// TIA Portal V17 export
// export: Created 2024-08-20T10:59:42.6043051Z, ExportSetting WithDefaults, DisplayName Totally Integrated Automation Portal, DisplayVersion V17 Update 4, DisplayName TIA Portal Openness, DisplayVersion V17 Update 4, DisplayName TIA Portal Version Control Interface, DisplayVersion V17, DisplayName STEP 7 Professional, DisplayVersion V17 Update 4, DisplayName STEP 7 Safety, DisplayVersion V17, DisplayName WinCC Advanced, DisplayVersion V17 Update 4
DATA_BLOCK "Redes"   // DB500
{ S7_Optimized_Access := 'FALSE' }
VERSION : 0.1
// stored: AutoNumber false, DBAccessibleFromOPCUA true, IsOnlyStoredInLoadMemory false, IsWriteProtectedInAS false
   VAR
      "CONNECT-MGE-PCM-E-CF-01" { S7_SetPoint := 'True'} : TCON_IP_v4;   // Dados de configuração
      "CONNECT-MGE-QGBT-AUX-01" { S7_SetPoint := 'True'} : TCON_IP_v4;   // Dados de configuração
      "Register-MGE-PCM-E-CF-01" : Array[0..38] of DInt;   // Tabela para receber os dados
      "Register-MGE-QGBT-AUX-01" : Array[0..38] of DInt;   // Tabela para receber os dados
      LADDR_PROFINET : HW_IOSYSTEM := 261;   // Endereço de hardware
      MODE_PROFINET : UInt := 4;   // Modo de operação da funcção
      RET_VAL_PROFINET : Int;   // Terorno de diagnóstico
      ESTADO_PROFINET : Array[0..1023] of Bool;   // Diagnóstico da rede PROFINET
      DONE_MB : Array[0..60] of Bool;   // Sinaliza fim de execução
      BUSY_MB : Array[0..60] of Bool;   // Sinaliza espera
      ERROR_MB : Array[0..60] of Bool;   // Sinaliza erro
      STATUS_MB : Array[0..60] of Word;   // Satus da comunicação
      START_MB : Array[0..60] of Bool;   // Inicia comunicação
      FCOM_MB : Array[0..60] of Bool;   // Falha de comunicação
      HAB_MB : Array[0..60] of Bool;   // Habilita comunicação MODBUS
      INICIA_MB : Bool;   // INICIA CICLO DE COMUNICAÇÃO MODBUS
      INI_AUX_MB : Bool;   // AUXILIAR DE INICIALIZAÇÃO
   END_VAR
BEGIN
   "CONNECT-MGE-PCM-E-CF-01".InterfaceId := 64;
   "CONNECT-MGE-PCM-E-CF-01".ID := 10;
   "CONNECT-MGE-PCM-E-CF-01".ConnectionType := 11;
   "CONNECT-MGE-PCM-E-CF-01".ActiveEstablished := TRUE;
   "CONNECT-MGE-PCM-E-CF-01".RemoteAddress.ADDR[1] := 192;
   "CONNECT-MGE-PCM-E-CF-01".RemoteAddress.ADDR[2] := 168;
   "CONNECT-MGE-PCM-E-CF-01".RemoteAddress.ADDR[3] := 2;
   "CONNECT-MGE-PCM-E-CF-01".RemoteAddress.ADDR[4] := 59;
   "CONNECT-MGE-PCM-E-CF-01".RemotePort := 502;
   "CONNECT-MGE-PCM-E-CF-01".LocalPort := 0;
   "CONNECT-MGE-QGBT-AUX-01".InterfaceId := 64;
   "CONNECT-MGE-QGBT-AUX-01".ID := 10;
   "CONNECT-MGE-QGBT-AUX-01".ConnectionType := 11;
   "CONNECT-MGE-QGBT-AUX-01".ActiveEstablished := TRUE;
   "CONNECT-MGE-QGBT-AUX-01".RemoteAddress.ADDR[1] := 192;
   "CONNECT-MGE-QGBT-AUX-01".RemoteAddress.ADDR[2] := 168;
   "CONNECT-MGE-QGBT-AUX-01".RemoteAddress.ADDR[3] := 2;
   "CONNECT-MGE-QGBT-AUX-01".RemoteAddress.ADDR[4] := 59;
   "CONNECT-MGE-QGBT-AUX-01".RemotePort := 502;
   "CONNECT-MGE-QGBT-AUX-01".LocalPort := 0;
   // "Register-MGE-PCM-E-CF-01"[0] : Tensão (L-N) fase 1
   // "Register-MGE-PCM-E-CF-01"[1] : Tensão (L-L) fase 1-2
   // "Register-MGE-PCM-E-CF-01"[2] : Corrente fase 1
   // "Register-MGE-PCM-E-CF-01"[3] : Cos φ fase 1
   // "Register-MGE-PCM-E-CF-01"[4] : Fator de potencia fase 1
   // "Register-MGE-PCM-E-CF-01"[5] : Potencia ativa fase 1
   // "Register-MGE-PCM-E-CF-01"[6] : Potência reativa fase 1
   // "Register-MGE-PCM-E-CF-01"[7] : Potência aparente fase 1
   // "Register-MGE-PCM-E-CF-01"[8] : THDV fase 1
   // "Register-MGE-PCM-E-CF-01"[9] : THDI fase 1
   // "Register-MGE-PCM-E-CF-01"[10] : Tensão (L-N) fase 2
   // "Register-MGE-PCM-E-CF-01"[11] : Tensão (L-L) fase 2-3
   // "Register-MGE-PCM-E-CF-01"[12] : Corrente fase 2
   // "Register-MGE-PCM-E-CF-01"[13] : Cos φ fase 2
   // "Register-MGE-PCM-E-CF-01"[14] : Fator de potência fase 2
   // "Register-MGE-PCM-E-CF-01"[15] : Potência ativa fase 2
   // "Register-MGE-PCM-E-CF-01"[16] : Potência reativa fase 2
   // "Register-MGE-PCM-E-CF-01"[17] : Potência aparente fase 2
   // "Register-MGE-PCM-E-CF-01"[18] : THDV fase 2
   // "Register-MGE-PCM-E-CF-01"[19] : THDI fase 2
   // "Register-MGE-PCM-E-CF-01"[20] : Tensão (L-N) fase 3
   // "Register-MGE-PCM-E-CF-01"[21] : Tensão (L-L) fase 3-1
   // "Register-MGE-PCM-E-CF-01"[22] : Corrente fase 3
   // "Register-MGE-PCM-E-CF-01"[23] : Cos φ fase 3
   // "Register-MGE-PCM-E-CF-01"[24] : Fator de potência fase 3
   // "Register-MGE-PCM-E-CF-01"[25] : Potência ativa fase 3
   // "Register-MGE-PCM-E-CF-01"[26] : Potência reativa fase 3
   // "Register-MGE-PCM-E-CF-01"[27] : Potência aparente fase 3
   // "Register-MGE-PCM-E-CF-01"[28] : THDV fase 3
   // "Register-MGE-PCM-E-CF-01"[29] : THDI fase 3
   // "Register-MGE-PCM-E-CF-01"[30] : Tensão média (L-N)
   // "Register-MGE-PCM-E-CF-01"[31] : Tensão média (L-L)
   // "Register-MGE-PCM-E-CF-01"[32] : Corrente total
   // "Register-MGE-PCM-E-CF-01"[33] : Fator de potência do sistema
   // "Register-MGE-PCM-E-CF-01"[34] : Potência ativa total
   // "Register-MGE-PCM-E-CF-01"[35] : Potência reativa total
   // "Register-MGE-PCM-E-CF-01"[36] : Potência aparente total
   // "Register-MGE-PCM-E-CF-01"[37] : Frequência do sistema
   // "Register-MGE-PCM-E-CF-01"[38] : Corrente de neutro
   // "Register-MGE-QGBT-AUX-01"[0] : Tensão (L-N) fase 1
   // "Register-MGE-QGBT-AUX-01"[1] : Tensão (L-L) fase 1-2
   // "Register-MGE-QGBT-AUX-01"[2] : Corrente fase 1
   // "Register-MGE-QGBT-AUX-01"[3] : Cos φ fase 1
   // "Register-MGE-QGBT-AUX-01"[4] : Fator de potencia fase 1
   // "Register-MGE-QGBT-AUX-01"[5] : Potencia ativa fase 1
   // "Register-MGE-QGBT-AUX-01"[6] : Potência reativa fase 1
   // "Register-MGE-QGBT-AUX-01"[7] : Potência aparente fase 1
   // "Register-MGE-QGBT-AUX-01"[8] : THDV fase 1
   // "Register-MGE-QGBT-AUX-01"[9] : THDI fase 1
   // "Register-MGE-QGBT-AUX-01"[10] : Tensão (L-N) fase 2
   // "Register-MGE-QGBT-AUX-01"[11] : Tensão (L-L) fase 2-3
   // "Register-MGE-QGBT-AUX-01"[12] : Corrente fase 2
   // "Register-MGE-QGBT-AUX-01"[13] : Cos φ fase 2
   // "Register-MGE-QGBT-AUX-01"[14] : Fator de potência fase 2
   // "Register-MGE-QGBT-AUX-01"[15] : Potência ativa fase 2
   // "Register-MGE-QGBT-AUX-01"[16] : Potência reativa fase 2
   // "Register-MGE-QGBT-AUX-01"[17] : Potência aparente fase 2
   // "Register-MGE-QGBT-AUX-01"[18] : THDV fase 2
   // "Register-MGE-QGBT-AUX-01"[19] : THDI fase 2
   // "Register-MGE-QGBT-AUX-01"[20] : Tensão (L-N) fase 3
   // "Register-MGE-QGBT-AUX-01"[21] : Tensão (L-L) fase 3-1
   // "Register-MGE-QGBT-AUX-01"[22] : Corrente fase 3
   // "Register-MGE-QGBT-AUX-01"[23] : Cos φ fase 3
   // "Register-MGE-QGBT-AUX-01"[24] : Fator de potência fase 3
   // "Register-MGE-QGBT-AUX-01"[25] : Potência ativa fase 3
   // "Register-MGE-QGBT-AUX-01"[26] : Potência reativa fase 3
   // "Register-MGE-QGBT-AUX-01"[27] : Potência aparente fase 3
   // "Register-MGE-QGBT-AUX-01"[28] : THDV fase 3
   // "Register-MGE-QGBT-AUX-01"[29] : THDI fase 3
   // "Register-MGE-QGBT-AUX-01"[30] : Tensão média (L-N)
   // "Register-MGE-QGBT-AUX-01"[31] : Tensão média (L-L)
   // "Register-MGE-QGBT-AUX-01"[32] : Corrente total
   // "Register-MGE-QGBT-AUX-01"[33] : Fator de potência do sistema
   // "Register-MGE-QGBT-AUX-01"[34] : Potência ativa total
   // "Register-MGE-QGBT-AUX-01"[35] : Potência reativa total
   // "Register-MGE-QGBT-AUX-01"[36] : Potência aparente total
   // "Register-MGE-QGBT-AUX-01"[37] : Frequência do sistema
   // "Register-MGE-QGBT-AUX-01"[38] : Corrente de neutro
END_DATA_BLOCK
